Staubli VAL3: _Chessie.pjx

--- _Chessie.pjx ---
Parameters version=s7.9 stackSize=5000 millimeterUnit=true
Program file=dataAcquisition.pgx
Program file=goToPoint.pgx
Program file=start.pgx
Program file=stop.pgx
Data file=_Chessie.dtx

--- goToPoint.pgx ---
program goToPoint()
begin
  logMsg("  goToPoint start")

  if(bPinceOpen == true)
    open(tTool)
  else
    close(tTool)
  endIf


  movel(pTarget, tTool, mRapide100)

  waitEndMove()

  bAcquisitionOk = false
end
